PROGRAM MAIN
VAR
	{attribute 'analysis' := '-33'}
	fbRpcServer : FB_RpcServer;
END_VAR

END_PROGRAM

(* stored: Version 1.1.0.1, ProductVersion 3.1.4024.12
   POU MAIN: Id {c5baf770-4e6d-4c1a-ac95-8140def6c61c}, SpecialFunc None *)
